TYPE "Positioning_MOL_Machine_Wng"
VERSION : 0.1
// Block: Positioning_MOL_Machine_Wng
   STRUCT
      NotAutReady : Bool;
      Minus_CndMissing : Bool;
      Plus_CndMissing : Bool;
      Ax_NotHomed : Bool;
      Ax : OOAx_Wng;
   END_STRUCT;

END_TYPE
